{attribute 'qualified_only'}
VAR_GLOBAL
	iMainFrame : INT;
	iReM: INT;
	iPM	: INT;
END_VAR

(* stored: Version 1.1.0.1, ProductVersion 3.1.4024.12
   GVL G_HMI: Id {1f28405a-7fc1-4023-8e02-e5a4478b4d4e} *)
